TYPE ST_CanFrame8 :
STRUCT
    data : ARRAY[0..7] OF BYTE;
END_STRUCT
END_TYPE

(* stored: Version 1.1.0.1
   DUT ST_CanFrame8: Id {1931d4e3-b64b-4e57-b189-2b42001a34fa} *)
